(* IEC 61131-3 sources: Siemens-Repository/Batch process oefening/src/4. Devices layer, 4 files *)

(* ---- DevBase.st ---- *)
{namespace Dev}
CLASS DevBase
    VAR

        Name        : string;
        Description : string;
        ControlMode : eDevControlMode := eDevControlMode#rOff;
    END_VAR

    METHOD public GetName : string
        GetName := Name;
    END_METHOD
    METHOD public GetDescription : string
        GetDescription := Name;
    END_METHOD

   METHOD PROTECTED Init : INT
    VAR_INPUT
        SetName : string;
        SetDescription : String;
    END_VAR

    IF SetName = '' THEN
        Init := 100;
        return;
    END_IF;

    if SetDescription = '' THEN
        init := 100;
        RETURN;
    END_IF;

    Name        := SetName;
    Description := SetDescription;
    END_METHOD

    METHOD PROTECTED Exec : INT

        Exec := 0;
        return;
    END_Method
END_CLASS

(* ---- DevDigitalInput.st ---- *)
USING System.Timer;

{namespace Dev}
CLASS DevDigitalInput EXTENDS DevBase
    VAR
        Hmi : hmiDevDigitalInput;

        tonValueTimer   :   OnDelay;
        tofValueTimer   :   OffDelay;
    END_VAR

    METHOD PROTECTED OVERRIDE Init : INT
        VAR_INPUT
            SetName : STRING;
            SetDescription : STRING;
        END_VAR

        if SUPER.Init(SetName := SetName, SetDescription := SetDescription) > 0 THEN
            Init := 100;
            return;
        END_IF;

        ControlMode := eDevControlMode#rOff;
    END_METHOD

    METHOD PROTECTED Exec : INT
        VAR_INPUT
            iRawValue   :   BOOL;
        END_VAR
        VAR_OUTPUT
            qRawValue   :   BOOL;
            qValue      :   BOOL;
        END_VAR
        VAR_TEMP
            tValue      :   BOOL;
            tValue2     :   BOOL;
        END_VAR

        tonValueTimer(signal := iRawValue, output => tValue);
        tofValueTimer(signal := tValue, output => tValue2);

       CASE ControlMode OF
        eDevControlMode#rOff:;

        eDevControlMode#rManual:

            qValue:= hmi.rwForceValue;

        eDevControlMode#rAuto:

            qRawValue := iRawValue;

            IF hmi.rwIsInverted THEN
                qValue := NOT tValue2;
            ELSE
                qValue := tValue2;
            END_IF;
       END_CASE;

        SUPER.Exec();
    END_METHOD

END_CLASS

(* ---- DevDigitalOutput.st ---- *)
{namespace Dev}
CLASS DevDigitalOutput EXTENDS DevBase
    VAR
        Hmi : hmiDevDigitalInput;
    END_VAR

    METHOD PROTECTED OVERRIDE Init : INT
        VAR_INPUT
            SetName : STRING;
            SetDescription : STRING;
        END_VAR

        if SUPER.Init(SetName := SetName, SetDescription := SetDescription) > 0 THEN
            Init := 100;
            return;
        END_IF;
    END_METHOD

END_CLASS

(* ---- DevMechanicalValve.st ---- *)
{namespace Dev}
CLASS DevMechanicalValve EXTENDS DevBase
    VAR
        FbkOpen     : DevDigitalInput;
        FbkClosed   : DevDigitalInput;

        CmdOpen     : DevDigitalOutput;
    END_VAR

END_CLASS
